// Publishes test results into an xUnit compatible Xml file
FUNCTION_BLOCK FB_xUnitXmlPublisher EXTENDS FB_BaseStatic IMPLEMENTS I_TestResultLogger
VAR
    // Dependency injection via FB_Init
    TestResults : I_TestResults;

    // File access mode
    AccessMode : SysFile.ACCESS_MODE := SysFile.AM_WRITE_PLUS;

    File : FB_FileControl;
    Xml : FB_XMLControl;
    BufferInitialised : BOOL := FALSE;
    Buffer : ARRAY [0..(GVL_Param_TcUnit.XUnitBufferSize - 1)] OF BYTE;
    WritingTestSuiteResultNumber : UINT(1..GVL_Param_TcUnit.MaxNumberOfTestSuites);
    PublishTrigger : R_TRIG;
END_VAR

(*
    Deletes the former file (if it exists).
    Opens the file, writes the buffer and closes it.
*)
METHOD PRIVATE DeleteOpenWriteClose : SysFile.SysTypes.RTS_IEC_RESULT;
VAR
    WriteResult : SysFile.SysTypes.RTS_IEC_RESULT;
END_VAR
DeleteOpenWriteClose := SysDir.CmpErrors.Errors.ERR_OK;
IF Initialised() THEN
    // Delete may fail if file doesn't exist yet (first run) — not a real error
    DeleteOpenWriteClose := MAX(DeleteOpenWriteClose, File.Delete(Filename := GVL_Param_TcUnit.xUnitFilePath));
    // Track Open/Write/Close separately for trace — these are the real errors
    WriteResult := File.Open(Filename := GVL_Param_TcUnit.xUnitFilePath, FileAccessMode := AccessMode);
    WriteResult := MAX(WriteResult, File.Write(BufferPointer := ADR(Buffer), Xml.Length));
    WriteResult := MAX(WriteResult, File.Close());
    DeleteOpenWriteClose := MAX(DeleteOpenWriteClose, WriteResult);
ELSE
    WriteResult := SysDir.CmpErrors.Errors.ERR_NOBUFFER;
    DeleteOpenWriteClose := WriteResult;
END_IF;

IF WriteResult <> SysDir.CmpErrors.Errors.ERR_OK THEN
    TraceWithSeverity(
        Message := CONCAT('xUnit file I/O failure: ', GVL_Param_TcUnit.xUnitFilePath),
        Severity := Global.TcEventSeverity.Error);
END_IF;
END_METHOD

(*
    FB_Init is always available implicitly AND it is used primarily FOR initialization.
    The return value is not evaluated. For a specific influence, you can also declare the
    methods explicitly and provide additional code there with the standard initialization
    code. You can evaluate the return value.
*)
METHOD FB_Init: BOOL
VAR_INPUT
    bInitRetains: BOOL; // TRUE: the retain variables are initialized (reset warm / reset cold)
    bInCopyCode: BOOL;  // TRUE: the instance will be copied to the copy code afterward (online change)
    iTestResults : I_TestResults; // Interface dependency injection
END_VAR
// Set buffer and flag
Xml.SetBuffer(PointerToBuffer := ADR(Buffer), SizeOfBuffer := SIZEOF(Buffer));

// Set buffer initialised
BufferInitialised := TRUE;

// Set testresult interface
THIS^.TestResults := iTestResults;
END_METHOD

METHOD PRIVATE Initialised : BOOL
Initialised := THIS^.BufferInitialised;
END_METHOD

(*
    This method is responsible for the entire generation of the output file. 
    The output of the xml writer is NOT beautified.

    When new data is available, feel free to add it to the report
*)
METHOD PUBLIC LogTestSuiteResults
VAR
    UnitTestResults : REFERENCE TO ST_TestSuiteResults;
    CurrentSuiteNumber : UINT;
    CurrentTestCount : UINT;
END_VAR
VAR CONSTANT
    TEST_STATUS_SKIP : STRING := 'SKIP';
    TEST_STATUS_PASS : STRING := 'PASS';
    TEST_STATUS_FAIL : STRING := 'FAIL';
END_VAR
UnitTestResults REF= TestResults.GetTestSuiteResults();

// Only publish once if "GVL_Param_TcUnit.xUnitEnablePublish" is enabled and all test results are stored.
PublishTrigger(CLK := (TestResults.GetAreTestResultsAvailable() AND GVL_Param_TcUnit.xUnitEnablePublish));
IF PublishTrigger.Q THEN

    // <?xml version="1.0" encoding="UTF-8"?>
    Xml.WriteDocumentHeader(Header := '<?xml version="1.0" encoding="UTF-8"?>');

    // <testsuites>  ('disabled' removed 2026-07-18: an empty string breaks JUnit
    //  parsers expecting an integer; skipped counts carry the information)
    Xml.NewTag('testsuites');
    Xml.NewParameter('failures', UDINT_TO_STRING(UnitTestResults.NumberOfFailedTestCases));
    (* 'tests' is the TOTAL testcase count; the previous successful-only value was a bug *)
    Xml.NewParameter('tests', UDINT_TO_STRING(UnitTestResults.NumberOfTestCases));
    Xml.NewParameter('skipped', UDINT_TO_STRING(UnitTestResults.NumberOfSkippedTestCases));
    Xml.NewParameter('time', LREAL_TO_STRING(UnitTestResults.Duration));

    FOR CurrentSuiteNumber := 1 TO UnitTestResults.NumberOfTestSuites BY 1 DO
        // <testsuite>
        Xml.NewTag('testsuite');
        Xml.NewParameter('id', UINT_TO_STRING(UnitTestResults.TestSuiteResults[CurrentSuiteNumber].Identity));
        Xml.NewParameter('name', UnitTestResults.TestSuiteResults[CurrentSuiteNumber].name);
        Xml.NewParameter('tests', UINT_TO_STRING(UnitTestResults.TestSuiteResults[CurrentSuiteNumber].NumberOfTests));
        Xml.NewParameter('failures', UINT_TO_STRING(UnitTestResults.TestSuiteResults[CurrentSuiteNumber].NumberOfFailedTests));
        Xml.NewParameter('skipped', UINT_TO_STRING(UnitTestResults.TestSuiteResults[CurrentSuiteNumber].NumberOfSkippedTests));
        Xml.NewParameter('time', LREAL_TO_STRING(UnitTestResults.TestSuiteResults[CurrentSuiteNumber].Duration));

        FOR CurrentTestCount := 1 TO UnitTestResults.TestSuiteResults[CurrentSuiteNumber].NumberOfTests BY 1 DO
            // <testcase>
            Xml.NewTag('testcase');
            Xml.NewParameter('name', UnitTestResults.TestSuiteResults[CurrentSuiteNumber].TestCaseResults[CurrentTestCount].TestName);
            Xml.NewParameter('classname', UnitTestResults.TestSuiteResults[CurrentSuiteNumber].TestCaseResults[CurrentTestCount].TestClassName);
            Xml.NewParameter('time', LREAL_TO_STRING(UnitTestResults.TestSuiteResults[CurrentSuiteNumber].TestCaseResults[CurrentTestCount].Duration));

            IF UnitTestResults.TestSuiteResults[CurrentSuiteNumber].TestCaseResults[CurrentTestCount].TestIsFailed THEN
                Xml.NewParameter('status', TEST_STATUS_FAIL);
            ELSIF UnitTestResults.TestSuiteResults[CurrentSuiteNumber].TestCaseResults[CurrentTestCount].TestIsSkipped THEN
                Xml.NewParameter('status', TEST_STATUS_SKIP);
            ELSE
                Xml.NewParameter('status', TEST_STATUS_PASS);
            END_IF

            // Determine testcase fail, skip, or success
            IF UnitTestResults.TestSuiteResults[CurrentSuiteNumber].TestCaseResults[CurrentTestCount].FailureType <> E_AssertionType.Type_UNDEFINED THEN
                (* In case of fail
                    <failure message="Values differ" type="BYTE" />
                *)
                Xml.NewTag('failure');
                Xml.NewParameter('message', UnitTestResults.TestSuiteResults[CurrentSuiteNumber].TestCaseResults[CurrentTestCount].FailureMessage);
                Xml.NewParameter('type', F_AssertionTypeToString(UnitTestResults.TestSuiteResults[CurrentSuiteNumber].TestCaseResults[CurrentTestCount].FailureType));
                // Close failure tag
                Xml.CloseTag();
            ELSIF UnitTestResults.TestSuiteResults[CurrentSuiteNumber].TestCaseResults[CurrentTestCount].TestIsSkipped THEN
                (* JUnit consumers recognize a skipped testcase through a <skipped/>
                   child element, not a custom status attribute (kept for
                   backward compatibility) *)
                Xml.NewTag('skipped');
                Xml.CloseTag();
            ELSE
            // In case of success
            Xml.NewTagData('');

            END_IF
            // Close testcase tag
            Xml.CloseTag();

        END_FOR
        // Close testsuite tag
        Xml.CloseTag();

    END_FOR
    // Close testsuites
    Xml.CloseTag();

    // Delete, open, save and close the file
    DeleteOpenWriteClose();

    // Clear the internal buffer
    Xml.ClearBuffer();

    // Inform user
    GVL_TcUnit.AdsMessageQueue.WriteLog(MsgCtrlMask := ADSLOG_MSGTYPE_HINT,
                                        msgFmtStr := '%s',
                                        strArg := '| ==========TEST RESULTS EXPORTED===========');

    GVL_TcUnit.AdsMessageQueue.WriteLog(MsgCtrlMask := ADSLOG_MSGTYPE_HINT,
                                        msgFmtStr :=  '| Location: %s ',
                                        strArg := GVL_Param_TcUnit.xUnitFilePath);

    GVL_TcUnit.AdsMessageQueue.WriteLog(MsgCtrlMask := ADSLOG_MSGTYPE_HINT,
                                        MsgFmtStr := '%s',
                                        StrArg := '| ======================================');

    TraceWithSeverity(
        Message := CONCAT('xUnit XML exported to ', GVL_Param_TcUnit.xUnitFilePath),
        Severity := Global.TcEventSeverity.Info);
END_IF
END_METHOD

END_FUNCTION_BLOCK

(* stored: Version 1.1.0.1
   POU FB_xUnitXmlPublisher: Id {6597c0b3-0890-4d5d-8d3a-2d0d0b2355db}, SpecialFunc None
   Method DeleteOpenWriteClose: Id {84256533-6eb5-465b-b1e5-db6f61e2e6c3}
   Method FB_Init: Id {0f23c47b-7245-415e-b489-0ae429217263}
   Method Initialised: Id {dac11801-83e2-4726-b3a7-dcd7f73621e3}
   Method LogTestSuiteResults: Id {32c3ccd7-3470-4554-b54c-b3a0a6491553} *)
